FUNCTION_BLOCK A2X_2AX_TO_2X (* Composite FB for convert 2 AX to A2X *)
  (* Standard: 61499-2; Description: Copyright (c) 2024 HR Agrartechnik GmbH This program and the accompanying materials are made available under the terms of the Eclipse Public License 2.0 which is available at https://www.eclipse.org/legal/epl-2.0/ SPDX-License-Identifier: EPL-2.0 *)
  (* Version 1.0, 2024-04-24, Franz Höpfinger, HR Agrartechnik GmbH *)
  PACKAGE adapter::conversion::unidirectional;
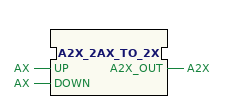
  SOCKETS
    UP : adapter::types::unidirectional::AX; (* TRUE = forward, up, right, clockwise *)
    DOWN : adapter::types::unidirectional::AX; (* TRUE = backward, down, left, counter-clockwise *)
  END_SOCKETS
  PLUGS
    A2X_OUT : adapter::types::unidirectional::A2X; (* Adapter Output *)
  END_PLUGS
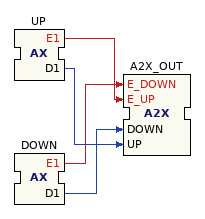
  EVENT_CONNECTIONS
    DOWN.E1 TO A2X_OUT.E_DOWN;
    UP.E1 TO A2X_OUT.E_UP;
  END_CONNECTIONS
  DATA_CONNECTIONS
    DOWN.D1 TO A2X_OUT.DOWN;
    UP.D1 TO A2X_OUT.UP;
  END_CONNECTIONS
END_FUNCTION_BLOCK
